// TIA Portal V19 export
DATA_BLOCK "IPC_Com_Channel_LOG_MACCHINA"   // DB191
// stored: MemoryReserve 100
   VAR
      SEND : Struct   // Invio singolo messaggio a MES
         ack : DInt;   // Acknowledge msg.ID From MES
         msg : "IPC_Msg_Generico";
      END_STRUCT;
   END_VAR
BEGIN
END_DATA_BLOCK
